FUNCTION_BLOCK ABSTRACT FB_AbstractFactory
VAR_INPUT
END_VAR
VAR_OUTPUT
END_VAR
VAR
END_VAR

METHOD M_GetColorObject : I_Color
VAR_INPUT
	eColor : E_Color;
END_VAR
END_METHOD

METHOD M_GetShapeObject : I_Shape
VAR_INPUT
	eShape : E_Shape;
END_VAR
END_METHOD

METHOD ABSTRACT M_ReleaseMemory : BOOL
VAR_INPUT
END_VAR
END_METHOD

END_FUNCTION_BLOCK

(* stored: Version 1.1.0.1, ProductVersion 3.1.4024.12
   POU FB_AbstractFactory: Id {7b35da90-6f2d-440c-8e0a-c1cc878589e6}, SpecialFunc None
   Method M_GetColorObject: Id {abc3931d-e852-4cd4-922d-47dd607a3800}
   Method M_GetShapeObject: Id {6bb60273-72dc-4375-937e-760f79af1d76}
   Method M_ReleaseMemory: Id {00a9ec82-33e2-42b7-be4b-78d65ff64f1e} *)
